// SIMATIC S7-200 SMART project (STEP 7-Micro/WIN SMART), CPU ST60

SYMBOL_TABLE V区符号
参数传输成功           V0.0     // 接收工控机传来的数据传输成功信号
参数是否更新           V0.1
挡板自动控制完成标志       V0.2
挡板电机开关           V0.3
挡板手动向内           V0.4
挡板手动向外           V0.5
置工件就绪            V0.6
下料电机开关           V0.7
下料前进点动           V1.0
下料后退点动           V1.1
冷却电机开关           V1.2
冷却电机向内           V1.3
冷却电机向外           V1.4
挡板查找原点完成标志       V1.5
挡板电机查找原点按钮       V11.1
下料电机查找原点按钮       V11.2
冷却电机查找原点按钮       V11.3
挡板自动控制           V11.4
下料下移一个工位         V11.5
下料启动按钮           V11.6
下料手动完成标志         V11.7
回到底部             V12.0
冷却自动控制           V12.1
挡板电机子例程          V20.1
挡板电机错误参数         VB21
挡板电机当前位置         VD24
挡板电机当前速度         VD28
挡板电机当前运动方向       V20.2
挡板电机移动位置         VD44
挡板电机速度           VD48
挡板电机移动模式         VB41
挡板电机停止运动轴        V40.1
挡板电机运动方向         V40.2
冷却电机子例程          V60.1
冷却电机错误参数         VB61
冷却电机当前位置         VD64
冷却电机当前速度         VD68
冷却电机当前运动方向       V60.2
冷却电机移动位置         VD84
冷却电机速度           VD88
冷却电机移动模式         VB81
冷却电机停止运动轴        V80.1
冷却电机运动方向         V80.2
下料电机子例程          V100.1
下料电机错误参数         VB101
下料电机当前位置         VD104
下料电机当前速度         VD108
下料电机当前运动方向       V100.2
下料电机移动位置         VD124
下料电机速度           VD128
下料电机移动模式         VB121
下料电机停止运动轴        V120.1
下料电机运动方向         V120.2
下料电机一号工位         VD150
下料电机杆件间距         VD154
下料电机二号工位         VD158
下料电机三号工位         VD162
下料电机四号工位         VD166
下料电机五号工位         VD170
下料电机取小车处         VD174
上一杆件数据           VD140
当前杆件数据           VD144
END_SYMBOL_TABLE

SYMBOL_TABLE 系统符号
Always_On        SM0.0    // 始终接通
END_SYMBOL_TABLE

SYMBOL_TABLE M区符号
挡板超限报警           M0.0     // 挡板的位置超过左右极限传感器的位置
更新配对表            M0.1
挡板步进到位状态位
电机是否就绪状态位        M0.3
上料步进到位状态位        M0.4
上料工件有无状态位        M0.5
下料步进到位状态位        M0.6
下料小车到位状态位        M0.7
步进报警信息           M1.0
上料传动故障报警         M1.1
上料杆件超限报警         M1.2
两次杆件之差           MD12
END_SYMBOL_TABLE

ORGANIZATION_BLOCK 程序块:OB1
TITLE=
BEGIN
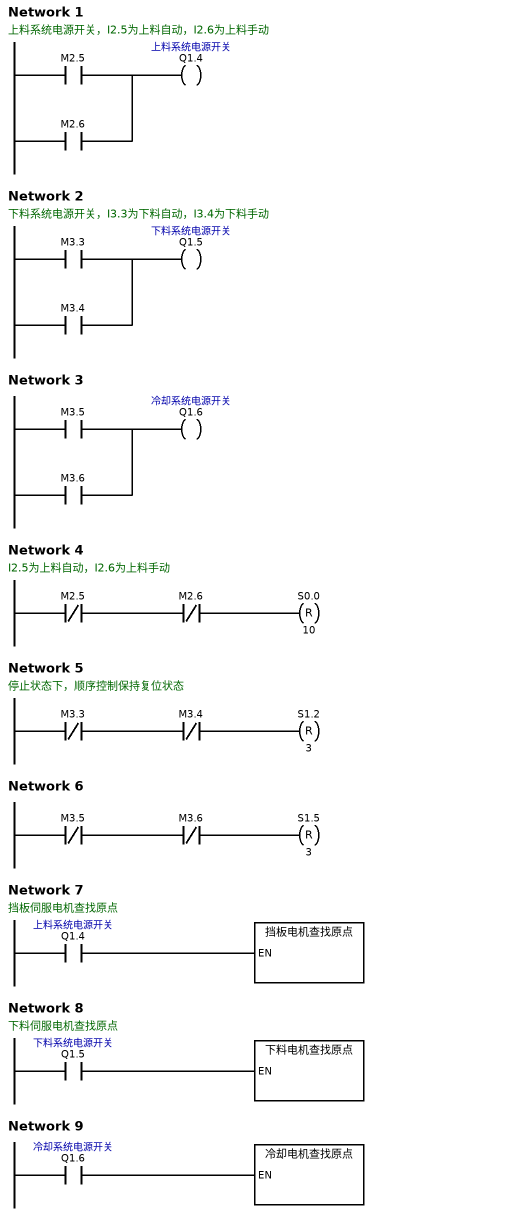
Network 1
// 上料系统电源开关，I2.5为上料自动，I2.6为上料手动
LD     M2.5
O      M2.6
=      上料系统电源开关:Q1.4
Network 2
// 下料系统电源开关，I3.3为下料自动，I3.4为下料手动
LD     M3.3
O      M3.4
=      下料系统电源开关:Q1.5
Network 3
LD     M3.5
O      M3.6
=      冷却系统电源开关:Q1.6
Network 4
// I2.5为上料自动，I2.6为上料手动
LDN    M2.5
AN     M2.6
R      S0.0, 10
Network 5
// 停止状态下，顺序控制保持复位状态
LDN    M3.3
AN     M3.4
R      S1.2, 3
Network 6
LDN    M3.5
AN     M3.6
R      S1.5, 3
Network 7
// 挡板伺服电机查找原点
LD     上料系统电源开关:Q1.4
CALL   挡板电机查找原点:SBR7
Network 8
// 下料伺服电机查找原点
LD     下料系统电源开关:Q1.5
CALL   下料电机查找原点:SBR0
Network 9
LD     冷却系统电源开关:Q1.6
CALL   冷却电机查找原点:SBR17
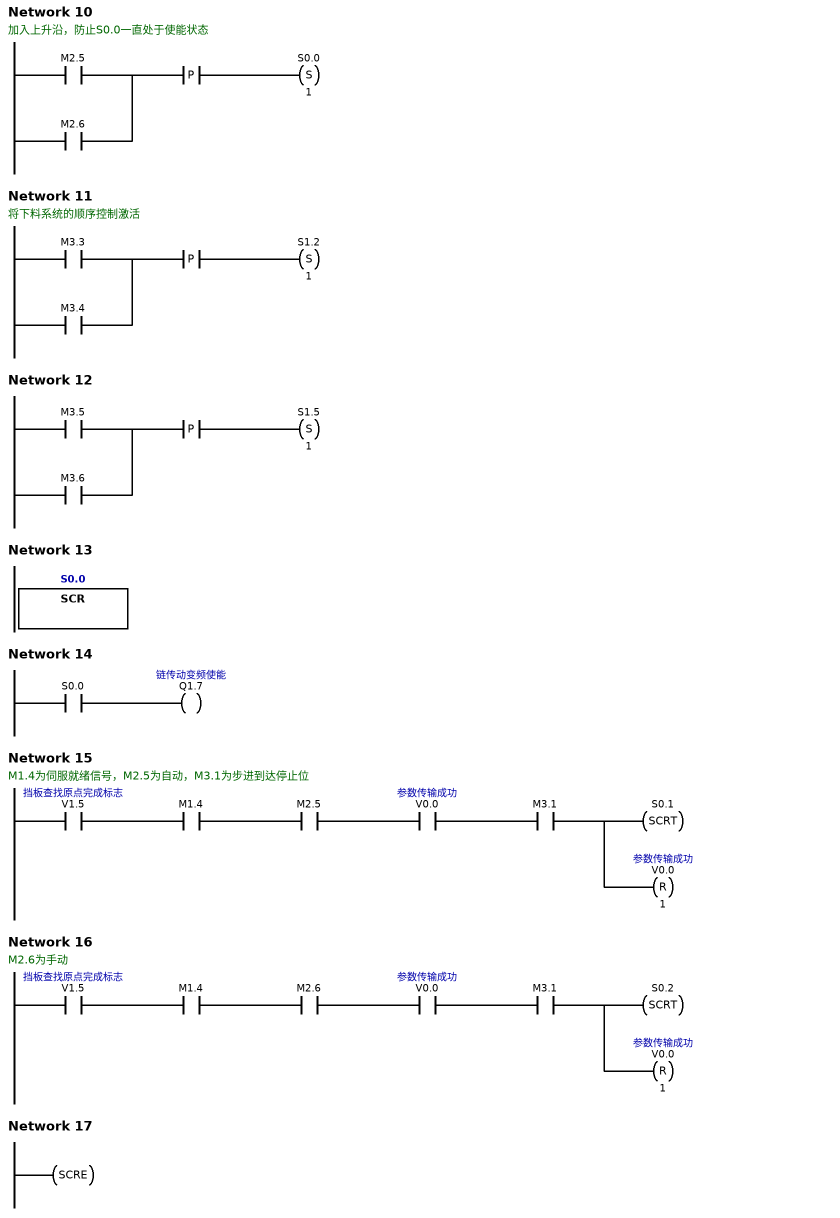
Network 10
// 加入上升沿，防止S0.0一直处于使能状态
LD     M2.5
O      M2.6
EU
S      S0.0, 1
Network 11
// 将下料系统的顺序控制激活
LD     M3.3
O      M3.4
EU
S      S1.2, 1
Network 12
LD     M3.5
O      M3.6
EU
S      S1.5, 1
Network 13
LSCR   S0.0
Network 14
LD     S0.0
=      链传动变频使能:Q1.7
Network 15
// M1.4为伺服就绪信号，M2.5为自动，M3.1为步进到达停止位
LD     挡板查找原点完成标志:V1.5
A      M1.4
A      M2.5
A      参数传输成功:V0.0
A      M3.1
SCRT   S0.1
R      参数传输成功:V0.0, 1
Network 16
// M2.6为手动
LD     挡板查找原点完成标志:V1.5
A      M1.4
A      M2.6
A      参数传输成功:V0.0
A      M3.1
SCRT   S0.2
R      参数传输成功:V0.0, 1
Network 17
SCRE
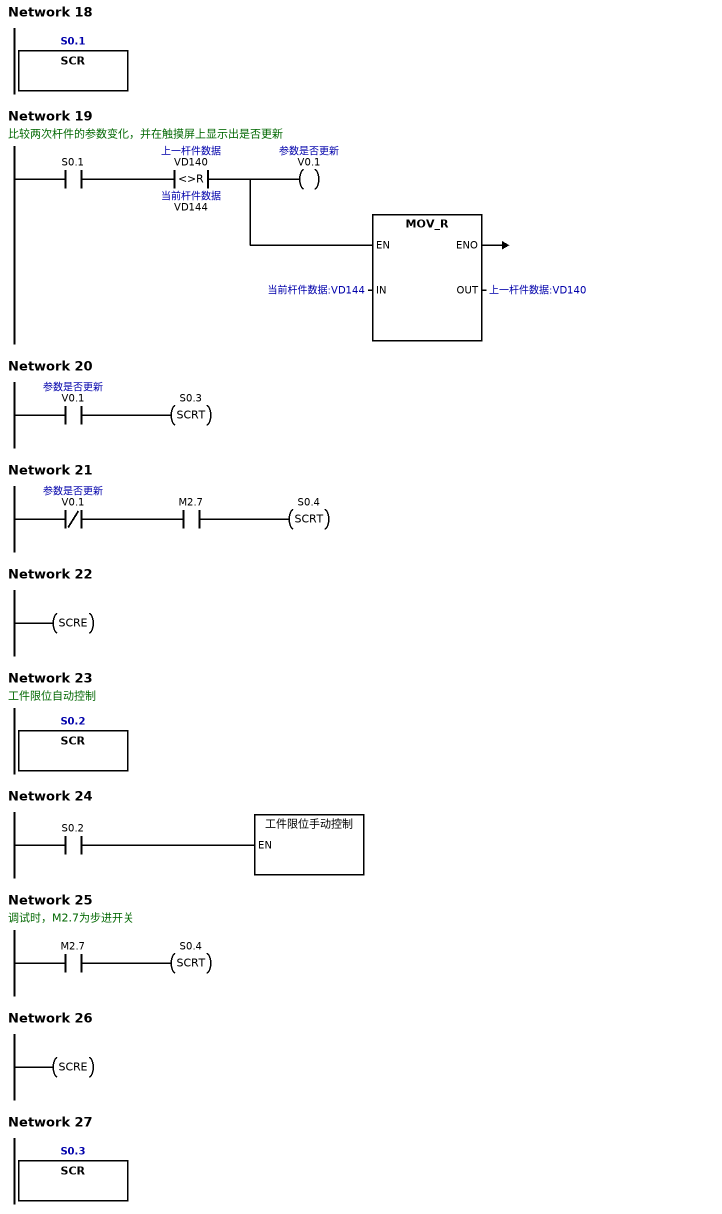
Network 18
LSCR   S0.1
Network 19
// 比较两次杆件的参数变化，并在触摸屏上显示出是否更新
LD     S0.1
AR<>   上一杆件数据:VD140, 当前杆件数据:VD144
=      参数是否更新:V0.1
MOVR   当前杆件数据:VD144, 上一杆件数据:VD140
Network 20
LD     参数是否更新:V0.1
SCRT   S0.3
Network 21
LDN    参数是否更新:V0.1
A      M2.7
SCRT   S0.4
Network 22
SCRE
Network 23
// 工件限位自动控制
LSCR   S0.2
Network 24
LD     S0.2
CALL   工件限位手动控制:SBR1
Network 25
// 调试时，M2.7为步进开关
LD     M2.7
SCRT   S0.4
Network 26
SCRE
Network 27
LSCR   S0.3
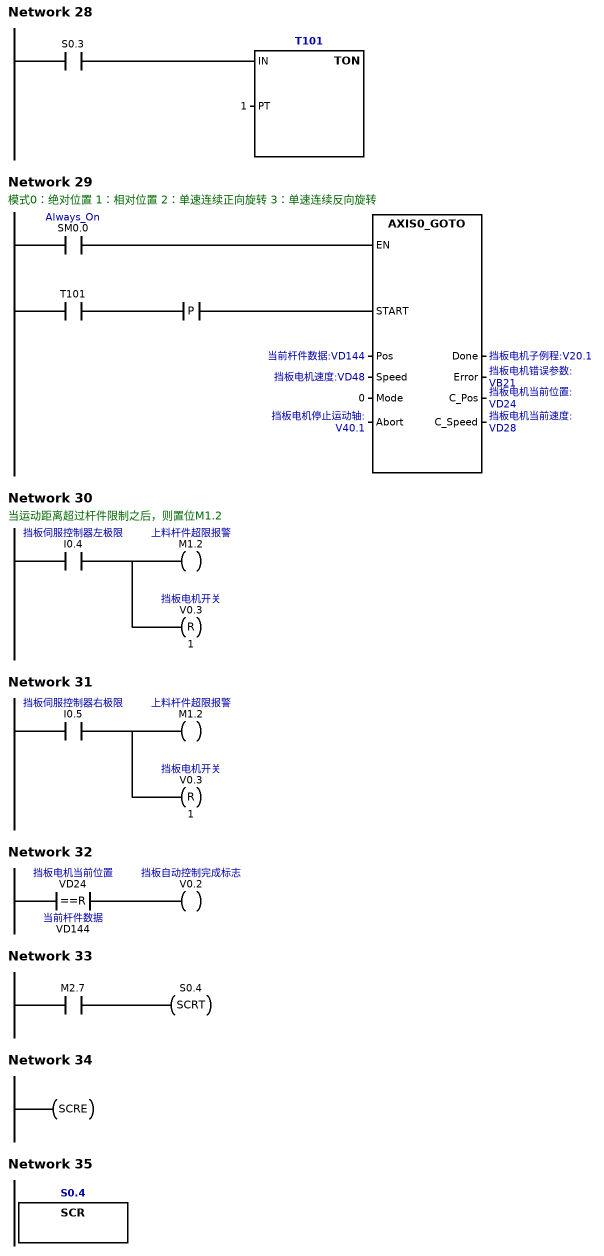
Network 28
LD     S0.3
TON    T101, 1
Network 29
// 模式0：绝对位置 1：相对位置 2：单速连续正向旋转 3：单速连续反向旋转
LD     Always_On:SM0.0
=      L60.0
LD     T101
EU
=      L63.7
LD     L60.0
CALL   AXIS0_GOTO:SBR4, L63.7, 当前杆件数据:VD144, 挡板电机速度:VD48, 0, 挡板电机停止运动轴:V40.1, 挡板电机子例程:V20.1, 挡板电机错误参数:VB21, 挡板电机当前位置:VD24, 挡板电机当前速度:VD28
Network 30
// 当运动距离超过杆件限制之后，则置位M1.2
LD     挡板伺服控制器左极限:I0.4
=      上料杆件超限报警:M1.2
R      挡板电机开关:V0.3, 1
Network 31
LD     挡板伺服控制器右极限:I0.5
=      上料杆件超限报警:M1.2
R      挡板电机开关:V0.3, 1
Network 32
LDR=   挡板电机当前位置:VD24, 当前杆件数据:VD144
=      挡板自动控制完成标志:V0.2
Network 33
LD     M2.7
SCRT   S0.4
Network 34
SCRE
Network 35
LSCR   S0.4
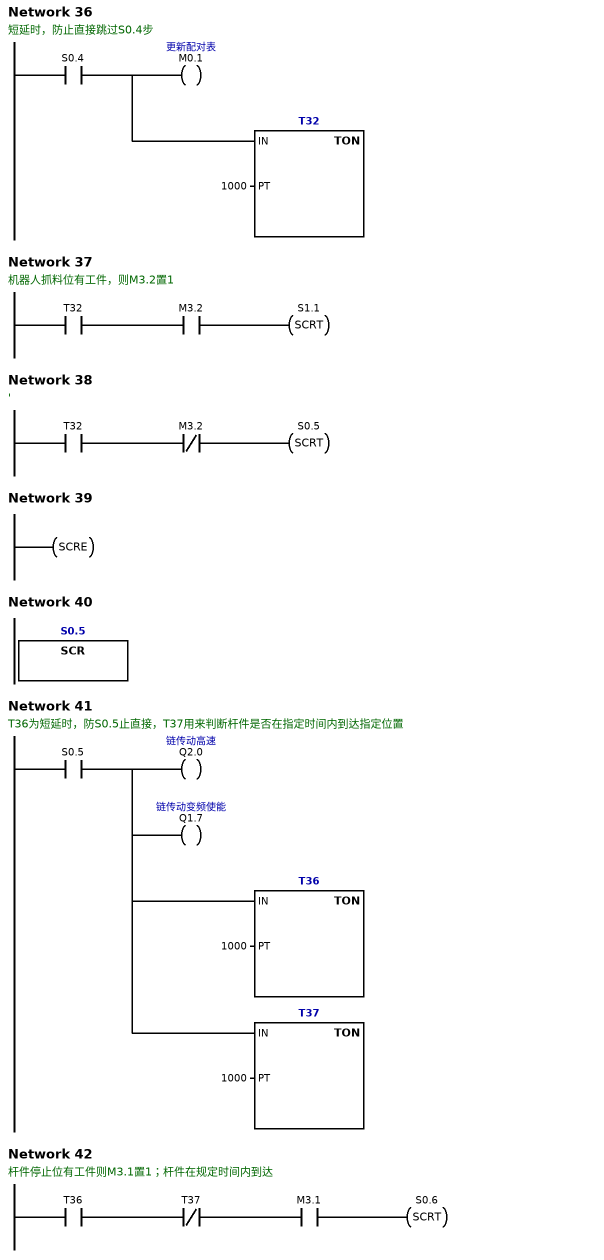
Network 36
// 短延时，防止直接跳过S0.4步
LD     S0.4
=      更新配对表:M0.1
TON    T32, 1000
Network 37
// 机器人抓料位有工件，则M3.2置1
LD     T32
A      M3.2
SCRT   S1.1
Network 38
// '
LD     T32
AN     M3.2
SCRT   S0.5
Network 39
SCRE
Network 40
LSCR   S0.5
Network 41
// T36为短延时，防S0.5止直接，T37用来判断杆件是否在指定时间内到达指定位置
LD     S0.5
=      链传动高速:Q2.0
=      链传动变频使能:Q1.7
TON    T36, 1000
TON    T37, 1000
Network 42
// 杆件停止位有工件则M3.1置1；杆件在规定时间内到达
LD     T36
AN     T37
A      M3.1
SCRT   S0.6
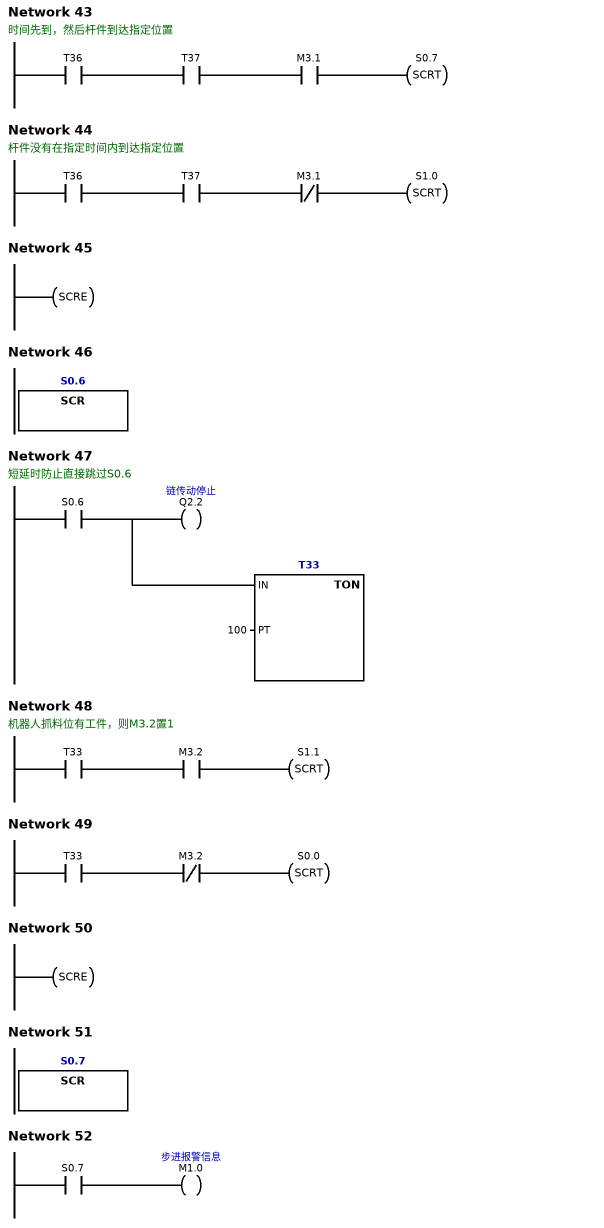
Network 43
// 时间先到，然后杆件到达指定位置
LD     T36
A      T37
A      M3.1
SCRT   S0.7
Network 44
// 杆件没有在指定时间内到达指定位置
LD     T36
A      T37
AN     M3.1
SCRT   S1.0
Network 45
SCRE
Network 46
LSCR   S0.6
Network 47
// 短延时防止直接跳过S0.6
LD     S0.6
=      链传动停止:Q2.2
TON    T33, 100
Network 48
// 机器人抓料位有工件，则M3.2置1
LD     T33
A      M3.2
SCRT   S1.1
Network 49
LD     T33
AN     M3.2
SCRT   S0.0
Network 50
SCRE
Network 51
LSCR   S0.7
Network 52
LD     S0.7
=      步进报警信息:M1.0
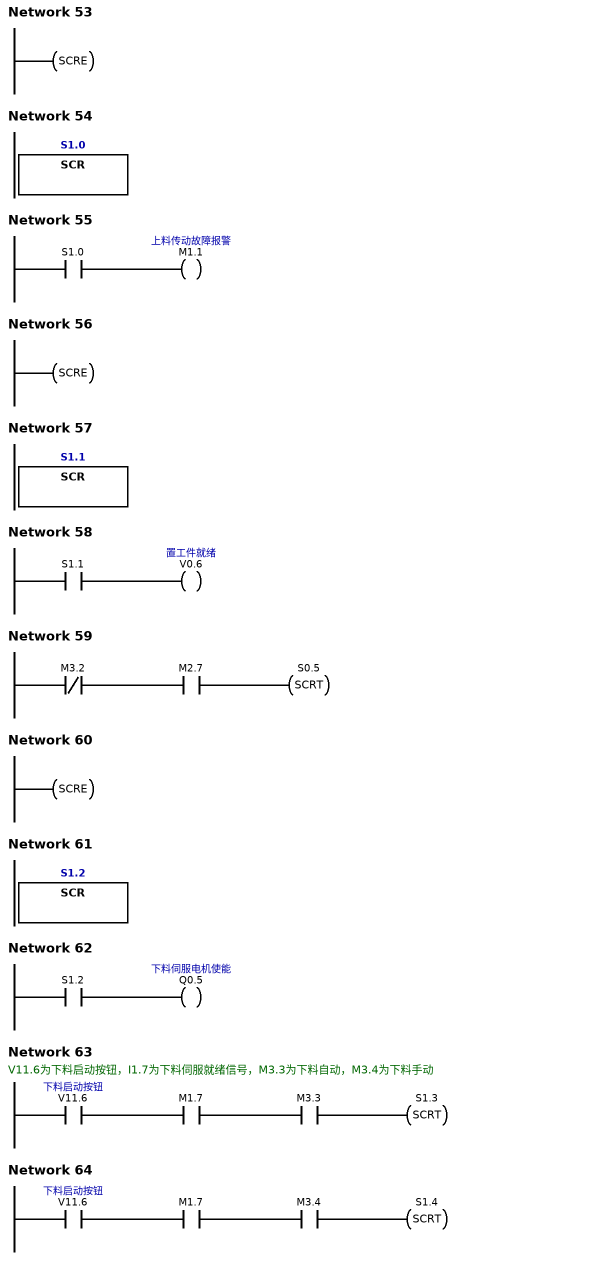
Network 53
SCRE
Network 54
LSCR   S1.0
Network 55
LD     S1.0
=      上料传动故障报警:M1.1
Network 56
SCRE
Network 57
LSCR   S1.1
Network 58
LD     S1.1
=      置工件就绪:V0.6
Network 59
LDN    M3.2
A      M2.7
SCRT   S0.5
Network 60
SCRE
Network 61
LSCR   S1.2
Network 62
LD     S1.2
=      下料伺服电机使能:Q0.5
Network 63
// V11.6为下料启动按钮，I1.7为下料伺服就绪信号，M3.3为下料自动，M3.4为下料手动
LD     下料启动按钮:V11.6
A      M1.7
A      M3.3
SCRT   S1.3
Network 64
LD     下料启动按钮:V11.6
A      M1.7
A      M3.4
SCRT   S1.4
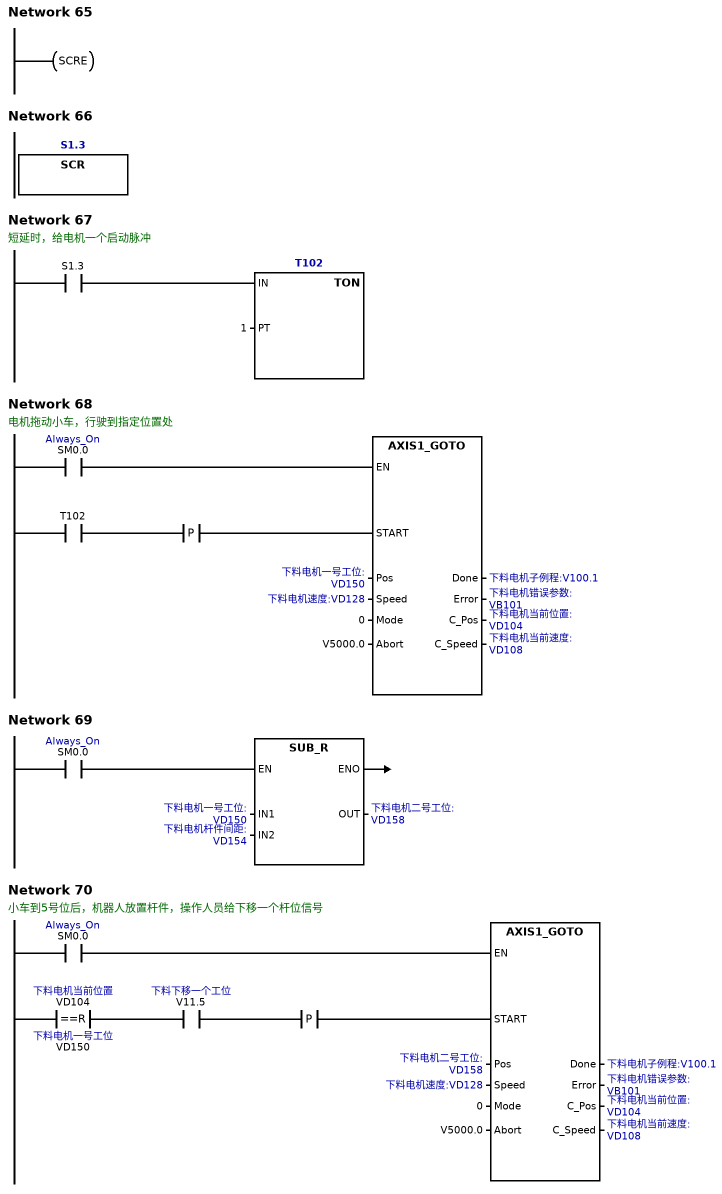
Network 65
SCRE
Network 66
LSCR   S1.3
Network 67
// 短延时，给电机一个启动脉冲
LD     S1.3
TON    T102, 1
Network 68
// 电机拖动小车，行驶到指定位置处
LD     Always_On:SM0.0
=      L60.0
LD     T102
EU
=      L63.7
LD     L60.0
CALL   AXIS1_GOTO:SBR11, L63.7, 下料电机一号工位:VD150, 下料电机速度:VD128, 0, V5000.0, 下料电机子例程:V100.1, 下料电机错误参数:VB101, 下料电机当前位置:VD104, 下料电机当前速度:VD108
Network 69
LD     Always_On:SM0.0
MOVR   下料电机一号工位:VD150, 下料电机二号工位:VD158
-R     下料电机杆件间距:VD154, 下料电机二号工位:VD158
Network 70
// 小车到5号位后，机器人放置杆件，操作人员给下移一个杆位信号
LD     Always_On:SM0.0
=      L60.0
LDR=   下料电机当前位置:VD104, 下料电机一号工位:VD150
A      下料下移一个工位:V11.5
EU
=      L63.7
LD     L60.0
CALL   AXIS1_GOTO:SBR11, L63.7, 下料电机二号工位:VD158, 下料电机速度:VD128, 0, V5000.0, 下料电机子例程:V100.1, 下料电机错误参数:VB101, 下料电机当前位置:VD104, 下料电机当前速度:VD108
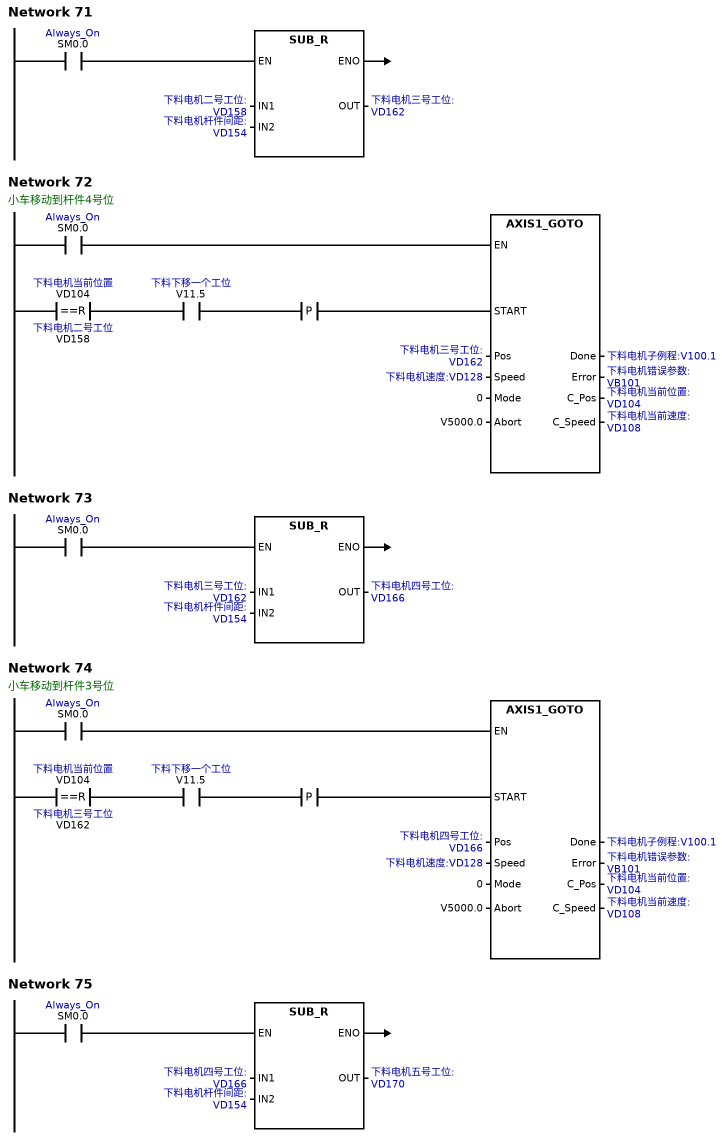
Network 71
LD     Always_On:SM0.0
MOVR   下料电机二号工位:VD158, 下料电机三号工位:VD162
-R     下料电机杆件间距:VD154, 下料电机三号工位:VD162
Network 72
// 小车移动到杆件4号位
LD     Always_On:SM0.0
=      L60.0
LDR=   下料电机当前位置:VD104, 下料电机二号工位:VD158
A      下料下移一个工位:V11.5
EU
=      L63.7
LD     L60.0
CALL   AXIS1_GOTO:SBR11, L63.7, 下料电机三号工位:VD162, 下料电机速度:VD128, 0, V5000.0, 下料电机子例程:V100.1, 下料电机错误参数:VB101, 下料电机当前位置:VD104, 下料电机当前速度:VD108
Network 73
LD     Always_On:SM0.0
MOVR   下料电机三号工位:VD162, 下料电机四号工位:VD166
-R     下料电机杆件间距:VD154, 下料电机四号工位:VD166
Network 74
// 小车移动到杆件3号位
LD     Always_On:SM0.0
=      L60.0
LDR=   下料电机当前位置:VD104, 下料电机三号工位:VD162
A      下料下移一个工位:V11.5
EU
=      L63.7
LD     L60.0
CALL   AXIS1_GOTO:SBR11, L63.7, 下料电机四号工位:VD166, 下料电机速度:VD128, 0, V5000.0, 下料电机子例程:V100.1, 下料电机错误参数:VB101, 下料电机当前位置:VD104, 下料电机当前速度:VD108
Network 75
LD     Always_On:SM0.0
MOVR   下料电机四号工位:VD166, 下料电机五号工位:VD170
-R     下料电机杆件间距:VD154, 下料电机五号工位:VD170
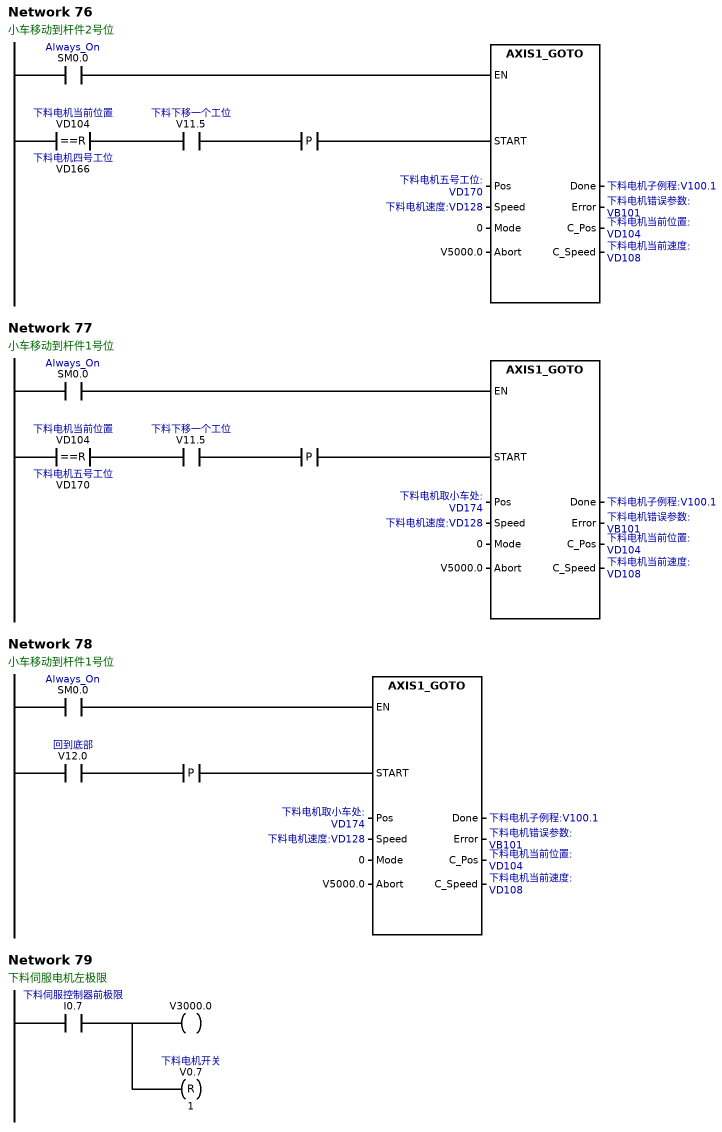
Network 76
// 小车移动到杆件2号位
LD     Always_On:SM0.0
=      L60.0
LDR=   下料电机当前位置:VD104, 下料电机四号工位:VD166
A      下料下移一个工位:V11.5
EU
=      L63.7
LD     L60.0
CALL   AXIS1_GOTO:SBR11, L63.7, 下料电机五号工位:VD170, 下料电机速度:VD128, 0, V5000.0, 下料电机子例程:V100.1, 下料电机错误参数:VB101, 下料电机当前位置:VD104, 下料电机当前速度:VD108
Network 77
// 小车移动到杆件1号位
LD     Always_On:SM0.0
=      L60.0
LDR=   下料电机当前位置:VD104, 下料电机五号工位:VD170
A      下料下移一个工位:V11.5
EU
=      L63.7
LD     L60.0
CALL   AXIS1_GOTO:SBR11, L63.7, 下料电机取小车处:VD174, 下料电机速度:VD128, 0, V5000.0, 下料电机子例程:V100.1, 下料电机错误参数:VB101, 下料电机当前位置:VD104, 下料电机当前速度:VD108
Network 78
// 小车移动到杆件1号位
LD     Always_On:SM0.0
=      L60.0
LD     回到底部:V12.0
EU
=      L63.7
LD     L60.0
CALL   AXIS1_GOTO:SBR11, L63.7, 下料电机取小车处:VD174, 下料电机速度:VD128, 0, V5000.0, 下料电机子例程:V100.1, 下料电机错误参数:VB101, 下料电机当前位置:VD104, 下料电机当前速度:VD108
Network 79
// 下料伺服电机左极限
LD     下料伺服控制器前极限:I0.7
=      V3000.0
R      下料电机开关:V0.7, 1
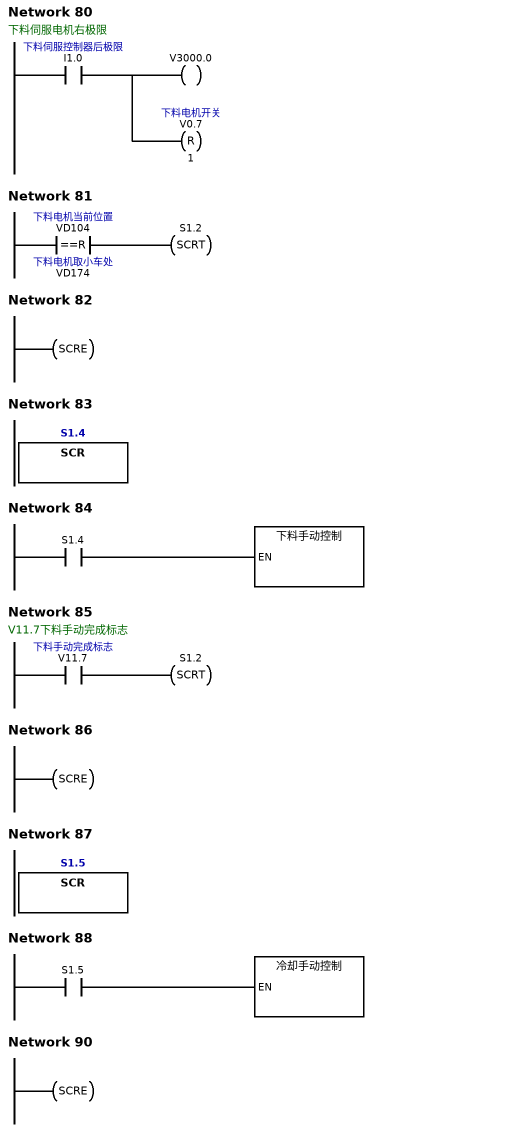
Network 80
// 下料伺服电机右极限
LD     下料伺服控制器后极限:I1.0
=      V3000.0
R      下料电机开关:V0.7, 1
Network 81
LDR=   下料电机当前位置:VD104, 下料电机取小车处:VD174
SCRT   S1.2
Network 82
SCRE
Network 83
LSCR   S1.4
Network 84
LD     S1.4
CALL   下料手动控制:SBR9
Network 85
// V11.7下料手动完成标志
LD     下料手动完成标志:V11.7
SCRT   S1.2
Network 86
SCRE
Network 87
LSCR   S1.5
Network 88
LD     S1.5
CALL   冷却手动控制:SBR18
Network 90
SCRE
END_ORGANIZATION_BLOCK

SUBROUTINE_BLOCK 下料电机查找原点:SBR0
TITLE=子程序注释
BEGIN
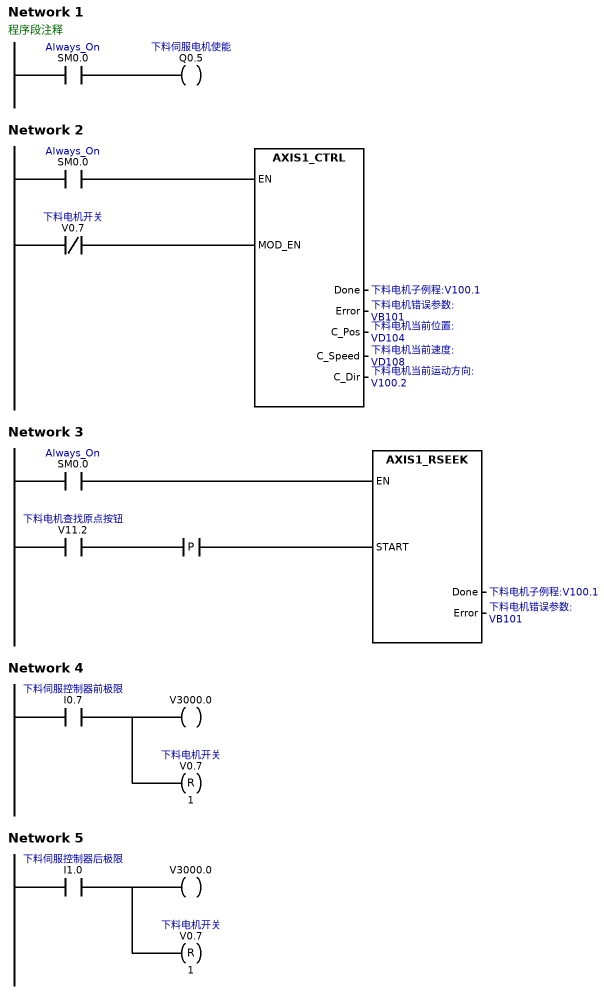
Network 1
// 程序段注释
LD     Always_On:SM0.0
=      下料伺服电机使能:Q0.5
Network 2
LD     Always_On:SM0.0
=      L60.0
LDN    下料电机开关:V0.7
=      L63.7
LD     L60.0
CALL   AXIS1_CTRL:SBR6, L63.7, 下料电机子例程:V100.1, 下料电机错误参数:VB101, 下料电机当前位置:VD104, 下料电机当前速度:VD108, 下料电机当前运动方向:V100.2
Network 3
LD     Always_On:SM0.0
=      L60.0
LD     下料电机查找原点按钮:V11.2
EU
=      L63.7
LD     L60.0
CALL   AXIS1_RSEEK:SBR12, L63.7, 下料电机子例程:V100.1, 下料电机错误参数:VB101
Network 4
LD     下料伺服控制器前极限:I0.7
=      V3000.0
R      下料电机开关:V0.7, 1
Network 5
LD     下料伺服控制器后极限:I1.0
=      V3000.0
R      下料电机开关:V0.7, 1
END_SUBROUTINE_BLOCK

SUBROUTINE_BLOCK 工件限位手动控制:SBR1
TITLE=子程序注释
BEGIN
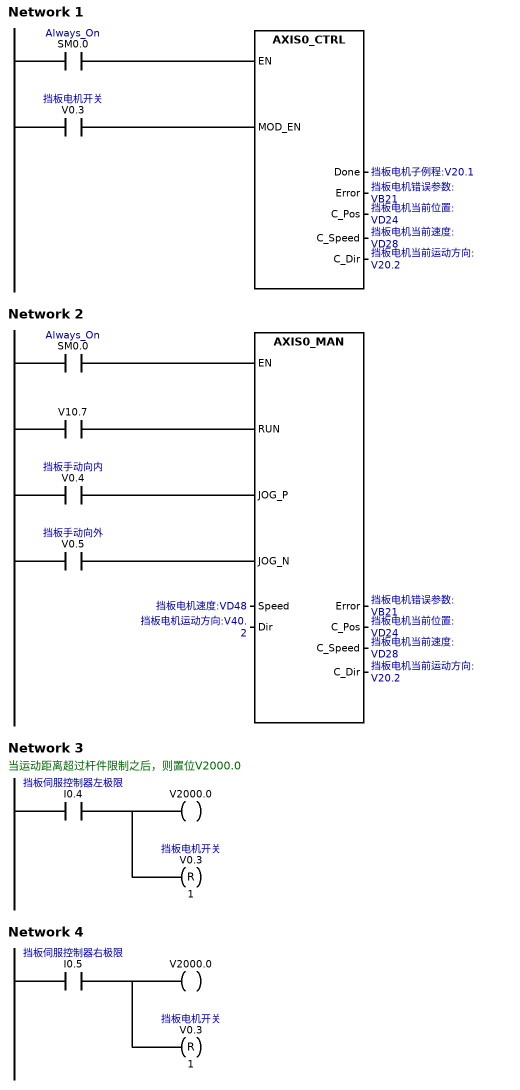
Network 1
LD     Always_On:SM0.0
=      L60.0
LD     挡板电机开关:V0.3
=      L63.7
LD     L60.0
CALL   AXIS0_CTRL:SBR2, L63.7, 挡板电机子例程:V20.1, 挡板电机错误参数:VB21, 挡板电机当前位置:VD24, 挡板电机当前速度:VD28, 挡板电机当前运动方向:V20.2
Network 2
LD     Always_On:SM0.0
=      L60.0
LD     V10.7
=      L63.7
LD     挡板手动向内:V0.4
=      L63.6
LD     挡板手动向外:V0.5
=      L63.5
LD     L60.0
CALL   AXIS0_MAN:SBR3, L63.7, L63.6, L63.5, 挡板电机速度:VD48, 挡板电机运动方向:V40.2, 挡板电机错误参数:VB21, 挡板电机当前位置:VD24, 挡板电机当前速度:VD28, 挡板电机当前运动方向:V20.2
Network 3
// 当运动距离超过杆件限制之后，则置位V2000.0
LD     挡板伺服控制器左极限:I0.4
=      V2000.0
R      挡板电机开关:V0.3, 1
Network 4
LD     挡板伺服控制器右极限:I0.5
=      V2000.0
R      挡板电机开关:V0.3, 1
END_SUBROUTINE_BLOCK

// SBR2: protected block, not included

// SBR3: protected block, not included

// SBR4: protected block, not included

// SBR5: protected block, not included

// SBR6: protected block, not included

SUBROUTINE_BLOCK 挡板电机查找原点:SBR7
TITLE=子程序注释
BEGIN
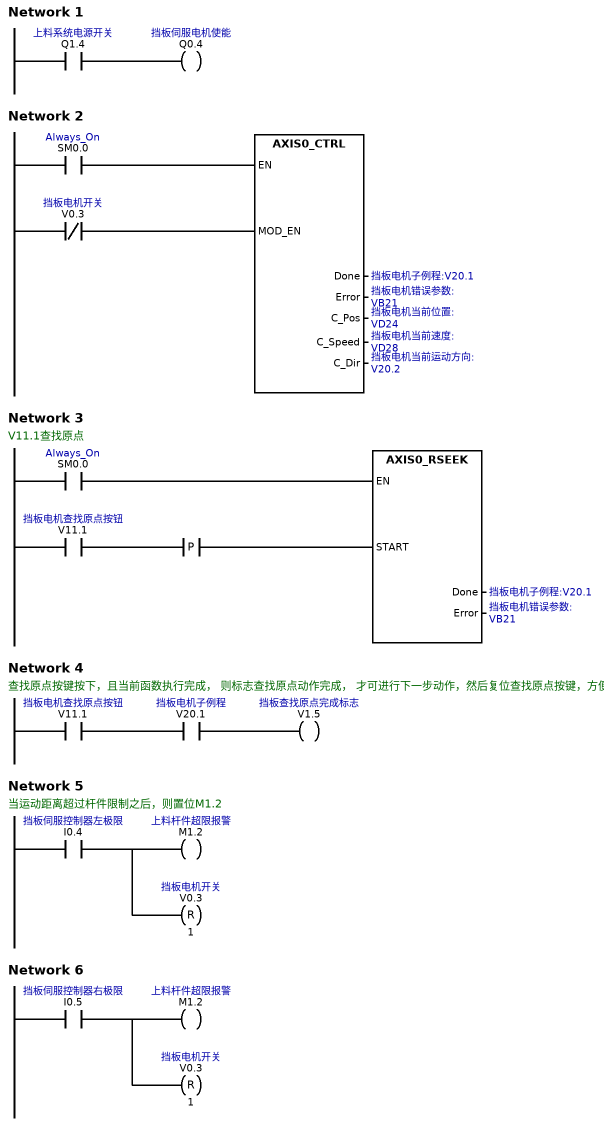
Network 1
LD     上料系统电源开关:Q1.4
=      挡板伺服电机使能:Q0.4
Network 2
LD     Always_On:SM0.0
=      L60.0
LDN    挡板电机开关:V0.3
=      L63.7
LD     L60.0
CALL   AXIS0_CTRL:SBR2, L63.7, 挡板电机子例程:V20.1, 挡板电机错误参数:VB21, 挡板电机当前位置:VD24, 挡板电机当前速度:VD28, 挡板电机当前运动方向:V20.2
Network 3
// V11.1查找原点
LD     Always_On:SM0.0
=      L60.0
LD     挡板电机查找原点按钮:V11.1
EU
=      L63.7
LD     L60.0
CALL   AXIS0_RSEEK:SBR5, L63.7, 挡板电机子例程:V20.1, 挡板电机错误参数:VB21
Network 4
// 查找原点按键按下，且当前函数执行完成， 则标志查找原点动作完成， 才可进行下一步动作，然后复位查找原点按键，方便下一次使用
LD     挡板电机查找原点按钮:V11.1
A      挡板电机子例程:V20.1
=      挡板查找原点完成标志:V1.5
Network 5
// 当运动距离超过杆件限制之后，则置位M1.2
LD     挡板伺服控制器左极限:I0.4
=      上料杆件超限报警:M1.2
R      挡板电机开关:V0.3, 1
Network 6
LD     挡板伺服控制器右极限:I0.5
=      上料杆件超限报警:M1.2
R      挡板电机开关:V0.3, 1
END_SUBROUTINE_BLOCK

SUBROUTINE_BLOCK 下料手动控制:SBR9
TITLE=子程序注释
BEGIN
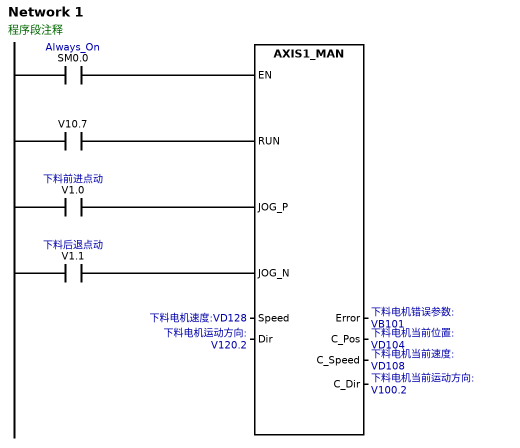
Network 1
// 程序段注释
LD     Always_On:SM0.0
=      L60.0
LD     V10.7
=      L63.7
LD     下料前进点动:V1.0
=      L63.6
LD     下料后退点动:V1.1
=      L63.5
LD     L60.0
CALL   AXIS1_MAN:SBR10, L63.7, L63.6, L63.5, 下料电机速度:VD128, 下料电机运动方向:V120.2, 下料电机错误参数:VB101, 下料电机当前位置:VD104, 下料电机当前速度:VD108, 下料电机当前运动方向:V100.2
END_SUBROUTINE_BLOCK

// SBR10: protected block, not included

// SBR11: protected block, not included

// SBR12: protected block, not included

// SBR13: protected block, not included

// SBR14: protected block, not included

// SBR15: protected block, not included

// SBR16: protected block, not included

SUBROUTINE_BLOCK 冷却电机查找原点:SBR17
TITLE=子程序注释
BEGIN
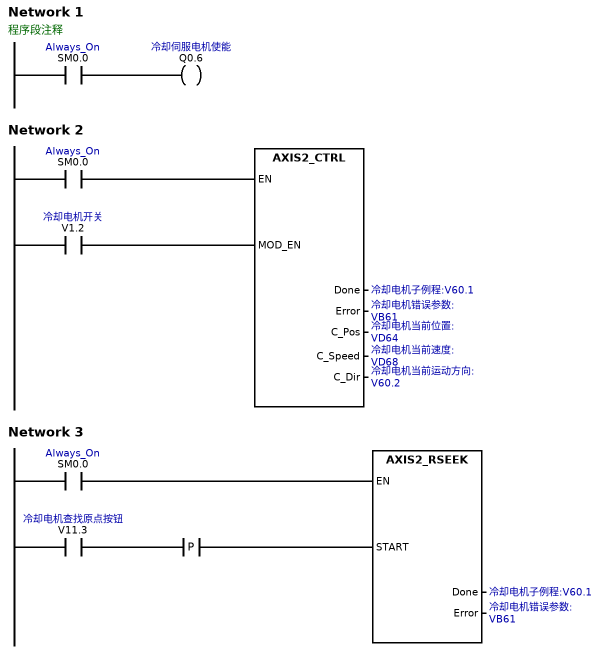
Network 1
// 程序段注释
LD     Always_On:SM0.0
=      冷却伺服电机使能:Q0.6
Network 2
LD     Always_On:SM0.0
=      L60.0
LD     冷却电机开关:V1.2
=      L63.7
LD     L60.0
CALL   AXIS2_CTRL:SBR13, L63.7, 冷却电机子例程:V60.1, 冷却电机错误参数:VB61, 冷却电机当前位置:VD64, 冷却电机当前速度:VD68, 冷却电机当前运动方向:V60.2
Network 3
LD     Always_On:SM0.0
=      L60.0
LD     冷却电机查找原点按钮:V11.3
EU
=      L63.7
LD     L60.0
CALL   AXIS2_RSEEK:SBR16, L63.7, 冷却电机子例程:V60.1, 冷却电机错误参数:VB61
END_SUBROUTINE_BLOCK

SUBROUTINE_BLOCK 冷却手动控制:SBR18
TITLE=子程序注释
BEGIN
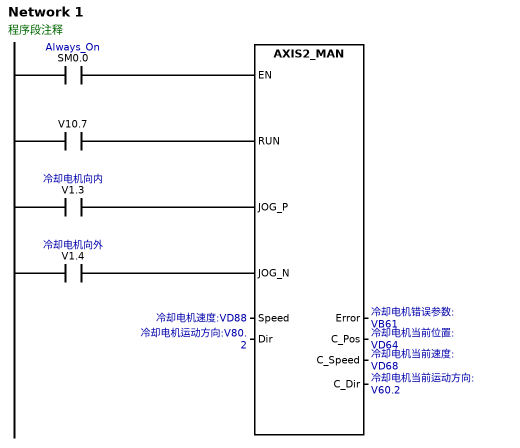
Network 1
// 程序段注释
LD     Always_On:SM0.0
=      L60.0
LD     V10.7
=      L63.7
LD     冷却电机向内:V1.3
=      L63.6
LD     冷却电机向外:V1.4
=      L63.5
LD     L60.0
CALL   AXIS2_MAN:SBR14, L63.7, L63.6, L63.5, 冷却电机速度:VD88, 冷却电机运动方向:V80.2, 冷却电机错误参数:VB61, 冷却电机当前位置:VD64, 冷却电机当前速度:VD68, 冷却电机当前运动方向:V60.2
END_SUBROUTINE_BLOCK
